Fanuc KAREL source: NC0074.KL

PROGRAM NC0074
%NOLOCKGROUP
ROUTINE R
VAR
  X : INTEGER
BEGIN
  X = 1
  WHILE X < 2 DO
    WHILE X < 2 DO
      WHILE X < 2 DO
        X = X + 1
      ENDWHILE
    ENDWHILE
  ENDWHILE
END R
BEGIN
  R
END NC0074
